ABB RobotStudio station: Session4.rspag

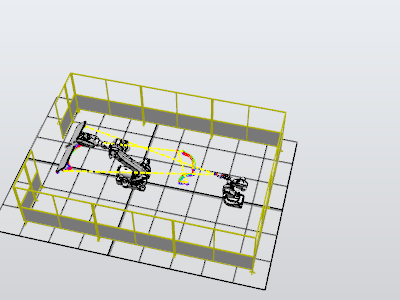
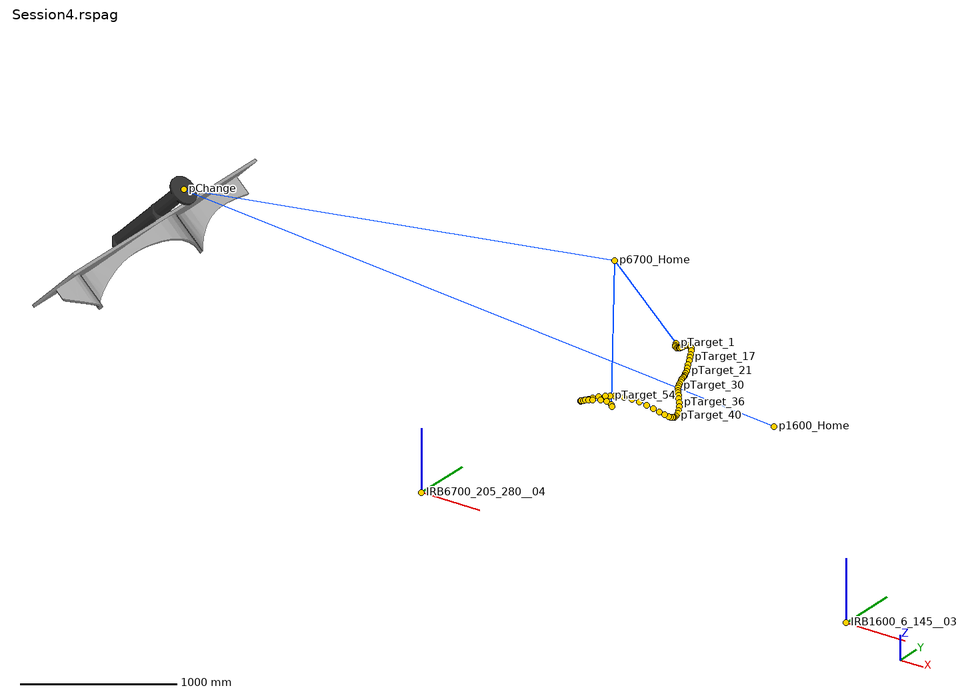
[picture v1: parts stored in the station drawn from their meshes, with robot base, taught points and paths (robot models come from the ABB library and are not in the file)]
--- station ---
Station Session4i (saved by RobotStudio 24.2.10821.1)
Controller Controller5, task T_ROB2: task frame (RAPID world) sits at (3300, 0, 0) mm, rotated rx 0 ry 0 rz 180 deg in the station
Controller Controller5, task T_ROB1: task frame (RAPID world) sits at (3300, 0, 0) mm, rotated rx 0 ry 0 rz 180 deg in the station
Controller Controller5
  mechanical unit ROB_1: IRB6700_205_280__04, 6 joints, base frame (3300, 0, 0) mm, rotated rx 0 ry 0 rz 180 deg
  mechanical unit ROB_2: IRB1600_6_145__03, 6 joints, base frame (0, 0, 0) mm
Layout (positions relative to the parent item):
  - IRB1600_6_145__03 [mechanism, from %ABB.RobotStudio.Models.IRB1600%\IRB1600_6_145_G_03.rslib] at (3300, 0, 0) mm, rotated rx 0 ry 0 rz 180 deg; joint values [0, -0.6981, 0.3491, 0, 0.4363, 3.1416] (rad or m)
  - IRB6700_205_280__04 [mechanism, from %ABB.RobotStudio.Models.IRB6700%\IRB6700_205_280__04.rslib] at (0, 0, 0) mm; joint values [0, -0.6981, -2.2689, 0, -0.9599, 0] (rad or m)
  - fence [graphiccomponentgroup, from Library\fence.rslib] at (-1500, 0, 0) mm
    - Fence_2500_1 [graphiccomponentgroup, from Equipment\Fence_2500.rslib] at (6000, 0, 0) mm
      - Body 1 [part, from Equipment\Fence_2500.rslib]
      - Body 2 [part, from Equipment\Fence_2500.rslib]
    - Fence_2500_2 [graphiccomponentgroup, from Equipment\Fence_2500.rslib] at (6000, -2500, 0) mm
      - Body 1 [part, from Equipment\Fence_2500.rslib]
      - Body 2 [part, from Equipment\Fence_2500.rslib]
    - Fence_2500_3 [graphiccomponentgroup, from Equipment\Fence_2500.rslib] at (6000, 2500, 0) mm, rotated rx 0 ry 0 rz 90 deg
      - Body 1 [part, from Equipment\Fence_2500.rslib]
      - Body 2 [part, from Equipment\Fence_2500.rslib]
    - Fence_2500_4 [graphiccomponentgroup, from Equipment\Fence_2500.rslib] at (6000, -2500, 0) mm, rotated rx 0 ry 0 rz 90 deg
      - Body 1 [part, from Equipment\Fence_2500.rslib]
      - Body 2 [part, from Equipment\Fence_2500.rslib]
    - Fence_2500_5 [graphiccomponentgroup, from Equipment\Fence_2500.rslib] at (3500, 2500, 0) mm, rotated rx 0 ry 0 rz 90 deg
      - Body 1 [part, from Equipment\Fence_2500.rslib]
      - Body 2 [part, from Equipment\Fence_2500.rslib]
    - Fence_2500_6 [graphiccomponentgroup, from Equipment\Fence_2500.rslib] at (3500, -2500, 0) mm, rotated rx 0 ry 0 rz 90 deg
      - Body 1 [part, from Equipment\Fence_2500.rslib]
      - Body 2 [part, from Equipment\Fence_2500.rslib]
    - Fence_2500_7 [graphiccomponentgroup, from Equipment\Fence_2500.rslib] at (1000, -2500, 0) mm, rotated rx 0 ry 0 rz 90 deg
      - Body 1 [part, from Equipment\Fence_2500.rslib]
      - Body 2 [part, from Equipment\Fence_2500.rslib]
    - Fence_2500_8 [graphiccomponentgroup, from Equipment\Fence_2500.rslib] at (1000, 2500, 0) mm, rotated rx 0 ry 0 rz 90 deg
      - Body 1 [part, from Equipment\Fence_2500.rslib]
      - Body 2 [part, from Equipment\Fence_2500.rslib]
    - Fence_Gate [graphiccomponentgroup, from Equipment\Fence_Gate.rslib] at (-1500, 2500, 0) mm, rotated rx 0 ry 0 rz 180 deg
      - Body 1 [part, from Equipment\Fence_Gate.rslib]
      - Body 2 [part, from Equipment\Fence_Gate.rslib]
      - Body 3 [part, from Equipment\Fence_Gate.rslib]
    - Fence_Gate_1 [graphiccomponentgroup, from Equipment\Fence_Gate.rslib] at (-1500, -1040, 0) mm, rotated rx 0 ry 0 rz 180 deg
      - Body 1 [part, from Equipment\Fence_Gate.rslib]
      - Body 2 [part, from Equipment\Fence_Gate.rslib]
      - Body 3 [part, from Equipment\Fence_Gate.rslib]
  - mySpintecTool [mechanism, from Library\mySpintecTool.rslib] at (2971.38, 0, 1222.28) mm, rotated rx -180 ry -85 rz 180 deg
  - training_part1 [part] at (-1843.45, 0, 1627.49) mm, rotated rx 180 ry -45 rz 180 deg, size 449.3 x 2022.8 x 720 mm
Attachment: mySpintecTool is attached to IRB1600_6_145__03 / Link6
Attachment: training_part1 is attached to IRB6700_205_280__04 / Link6
Targets, tools, work objects and paths stored in the station and not in the controller backup, written as RAPID:
! task T_ROB1
MODULE Module1
  VAR SyncIdent Ident_1;
  VAR SyncIdent Ident_2;
ENDMODULE

! task T_ROB2
MODULE Module1
  CONST robtarget Target_10:=[[-249.999367219,-2.759503933,70.911791319],[0.082627052,-0.189001665,0.896559115,0.391960322],[0,0,0,0],[9E+09,9E+09,9E+09,9E+09,9E+09,9E+09]];
  CONST robtarget Target_20:=[[-272.860994804,33.003713337,109.273686321],[0.078888886,-0.183345526,0.900091869,0.387292639],[0,0,0,0],[9E+09,9E+09,9E+09,9E+09,9E+09,9E+09]];
  CONST robtarget Target_30:=[[-293.909747151,69.703915361,146.790608764],[0.066447689,-0.162722707,0.911372094,0.372165194],[0,0,0,0],[9E+09,9E+09,9E+09,9E+09,9E+09,9E+09]];
  CONST robtarget Target_40:=[[-309.049057288,104.287364252,178.817535141],[0.044488261,-0.119397612,0.929423604,0.346318884],[0,0,0,0],[9E+09,9E+09,9E+09,9E+09,9E+09,9E+09]];
  CONST robtarget Target_50:=[[-315.82436696,131.079185384,200.514549492],[0.018847209,-0.056496391,0.946916759,0.315913899],[0,0,0,0],[9E+09,9E+09,9E+09,9E+09,9E+09,9E+09]];
  CONST robtarget Target_60:=[[-316.949093873,142.442010103,208.738875508],[0.005635439,-0.017961808,0.953951582,0.299369328],[0,0,0,0],[9E+09,9E+09,9E+09,9E+09,9E+09,9E+09]];
  CONST robtarget Target_70:=[[-316.981336532,150.771457316,214.363656376],[0.00472652,-0.015856219,-0.958220782,-0.285550649],[0,0,0,0],[9E+09,9E+09,9E+09,9E+09,9E+09,9E+09]];
  CONST robtarget Target_80:=[[-316.204048535,159.553535577,219.906336386],[0.015917508,-0.05682374,-0.961261763,-0.269246205],[0,0,0,0],[9E+09,9E+09,9E+09,9E+09,9E+09,9E+09]];
  CONST robtarget Target_90:=[[-312.751266422,174.803616127,228.540118146],[0.032209123,-0.130949879,-0.962189752,-0.236654987],[0,0,0,0],[9E+09,9E+09,9E+09,9E+09,9E+09,9E+09]];
  CONST robtarget Target_100:=[[-304.928487553,193.590972725,237.35167523],[0.043068547,-0.216929266,-0.956567695,-0.189907974],[0,0,0,0],[9E+09,9E+09,9E+09,9E+09,9E+09,9E+09]];
  CONST robtarget Target_110:=[[-295.35254505,209.582414865,243.17789314],[0.042988124,-0.279779228,-0.947977395,-0.145651859],[0,0,0,0],[9E+09,9E+09,9E+09,9E+09,9E+09,9E+09]];
  CONST robtarget Target_120:=[[-283.89767317,224.89172178,247.2508217],[0.035173025,-0.328290116,-0.938550871,-0.100552084],[0,0,0,0],[9E+09,9E+09,9E+09,9E+09,9E+09,9E+09]];
  CONST robtarget Target_130:=[[-263.239275575,247.748070357,250.552666299],[0.014250971,-0.37796017,-0.925055022,-0.034874436],[0,0,0,0],[9E+09,9E+09,9E+09,9E+09,9E+09,9E+09]];
  CONST robtarget Target_140:=[[-240.980203403,269.118585414,250.90982541],[0.007976683,0.402341156,0.915275131,-0.018149404],[0,0,0,0],[9E+09,9E+09,9E+09,9E+09,9E+09,9E+09]];
  CONST robtarget Target_150:=[[-208.411538431,298.031041245,247.790506063],[0.034910793,0.408676536,0.908701592,-0.077628235],[0,0,0,0],[9E+09,9E+09,9E+09,9E+09,9E+09,9E+09]];
  CONST robtarget Target_160:=[[-176.050652943,326.808930331,241.226021251],[0.053503703,0.389404955,0.910952455,-0.125166922],[0,0,0,0],[9E+09,9E+09,9E+09,9E+09,9E+09,9E+09]];
  CONST robtarget Target_170:=[[-156.251547721,345.811133404,235.321691527],[0.059919365,0.36278175,0.917514208,-0.151547844],[0,0,0,0],[9E+09,9E+09,9E+09,9E+09,9E+09,9E+09]];
  CONST robtarget Target_180:=[[-137.911367006,365.728959049,228.015632898],[0.060848306,0.321409713,0.928490022,-0.175782705],[0,0,0,0],[9E+09,9E+09,9E+09,9E+09,9E+09,9E+09]];
  CONST robtarget Target_190:=[[-123.074825841,385.296017373,219.901370788],[0.055303407,0.265093219,0.942346679,-0.196595667],[0,0,0,0],[9E+09,9E+09,9E+09,9E+09,9E+09,9E+09]];
  CONST robtarget Target_200:=[[-112.483952008,403.752551203,211.51909834],[0.044543145,0.199537763,0.95536135,-0.213272783],[0,0,0,0],[9E+09,9E+09,9E+09,9E+09,9E+09,9E+09]];
  CONST robtarget Target_210:=[[-105.66911776,420.539983076,203.415477486],[0.032817077,0.140384123,0.963573356,-0.225259238],[0,0,0,0],[9E+09,9E+09,9E+09,9E+09,9E+09,9E+09]];
  CONST robtarget Target_220:=[[-101.152730173,437.795026941,194.70341226],[0.02007137,0.08291124,0.968380047,-0.234441785],[0,0,0,0],[9E+09,9E+09,9E+09,9E+09,9E+09,9E+09]];
  CONST robtarget Target_230:=[[-99.0040493,453.549567144,186.489814416],[0.008561695,0.034579383,0.970065446,-0.240216557],[0,0,0,0],[9E+09,9E+09,9E+09,9E+09,9E+09,9E+09]];
  CONST robtarget Target_240:=[[-98.516394989,465.109909633,180.348088014],[0.000491395,0.001966291,0.970025575,-0.242994396],[0,0,0,0],[9E+09,9E+09,9E+09,9E+09,9E+09,9E+09]];
  CONST robtarget Target_250:=[[-98.913820285,477.215623072,173.84543664],[0.007456826,0.029529533,-0.969123936,0.244685919],[0,0,0,0],[9E+09,9E+09,9E+09,9E+09,9E+09,9E+09]];
  CONST robtarget Target_260:=[[-101.158760793,495.694459859,163.84647429],[0.018390599,0.072530228,-0.966611976,0.245076395],[0,0,0,0],[9E+09,9E+09,9E+09,9E+09,9E+09,9E+09]];
  CONST robtarget Target_270:=[[-106.104979829,517.566463562,152.024862353],[0.029263347,0.116194115,-0.962734999,0.242453924],[0,0,0,0],[9E+09,9E+09,9E+09,9E+09,9E+09,9E+09]];
  CONST robtarget Target_280:=[[-113.660346961,540.614341097,139.758405519],[0.038221783,0.154953239,-0.958456095,0.236411725],[0,0,0,0],[9E+09,9E+09,9E+09,9E+09,9E+09,9E+09]];
  CONST robtarget Target_290:=[[-130.507549693,578.661351825,120.440667817],[0.047524101,0.206136989,-0.952386495,0.2195654],[0,0,0,0],[9E+09,9E+09,9E+09,9E+09,9E+09,9E+09]];
  CONST robtarget Target_300:=[[-151.266393323,615.999238015,103.277260281],[0.050249688,0.24477104,-0.948497911,0.194714713],[0,0,0,0],[9E+09,9E+09,9E+09,9E+09,9E+09,9E+09]];
  CONST robtarget Target_310:=[[-176.02610459,654.710741932,88.198539481],[0.046456986,0.275583142,-0.946795556,0.159605309],[0,0,0,0],[9E+09,9E+09,9E+09,9E+09,9E+09,9E+09]];
  CONST robtarget Target_320:=[[-202.970542535,693.300547015,76.716257128],[0.035884116,0.297986116,-0.947053887,0.114041831],[0,0,0,0],[9E+09,9E+09,9E+09,9E+09,9E+09,9E+09]];
  CONST robtarget Target_330:=[[-231.602130589,732.417304287,69.542021834],[0.018589095,0.31143545,-0.948397291,0.056612584],[0,0,0,0],[9E+09,9E+09,9E+09,9E+09,9E+09,9E+09]];
  CONST robtarget Target_340:=[[-260.470210824,771.255251336,67.256102726],[0.000027118,0.313521967,-0.949580944,0.000077659],[0,0,0,0],[9E+09,9E+09,9E+09,9E+09,9E+09,9E+09]];
  CONST robtarget Target_350:=[[-291.671653455,813.968299538,69.78080258],[0.017514958,-0.303598774,0.9510575,0.054869325],[0,0,0,0],[9E+09,9E+09,9E+09,9E+09,9E+09,9E+09]];
  CONST robtarget Target_360:=[[-321.100482584,856.495332628,76.875137674],[0.030055142,-0.282317538,0.953462043,0.101506791],[0,0,0,0],[9E+09,9E+09,9E+09,9E+09,9E+09,9E+09]];
  CONST robtarget Target_370:=[[-347.608236851,898.755866406,87.798617829],[0.03661292,-0.250273308,0.957292518,0.140049279],[0,0,0,0],[9E+09,9E+09,9E+09,9E+09,9E+09,9E+09]];
  CONST robtarget Target_380:=[[-370.0464549,940.669416672,101.810752862],[0.036758138,-0.206846372,0.962600213,0.171067961],[0,0,0,0],[9E+09,9E+09,9E+09,9E+09,9E+09,9E+09]];
  CONST robtarget Target_390:=[[-386.422870207,979.737745125,117.176024402],[0.030820624,-0.15395644,0.968381142,0.193869719],[0,0,0,0],[9E+09,9E+09,9E+09,9E+09,9E+09,9E+09]];
  CONST robtarget Target_400:=[[-397.441727713,1019.682361901,134.633461354],[0.01837918,-0.084776151,0.973609592,0.211091382],[0,0,0,0],[9E+09,9E+09,9E+09,9E+09,9E+09,9E+09]];
  CONST robtarget Target_410:=[[-400.68526788,1043.112626972,145.490242444],[0.008067365,-0.036072035,0.975216982,0.218141154],[0,0,0,0],[9E+09,9E+09,9E+09,9E+09,9E+09,9E+09]];
  CONST robtarget Target_420:=[[-401.329476368,1057.285914809,152.218968855],[0.000811987,-0.00358584,0.975219049,0.221210962],[0,0,0,0],[9E+09,9E+09,9E+09,9E+09,9E+09,9E+09]];
  CONST robtarget Target_430:=[[-400.962720054,1070.625724022,158.636236091],[0.006312666,-0.02754754,-0.974356125,-0.223229532],[0,0,0,0],[9E+09,9E+09,9E+09,9E+09,9E+09,9E+09]];
  CONST robtarget Target_440:=[[-398.849530954,1089.506582954,167.817808857],[0.016104926,-0.069657841,-0.97181004,-0.224663442],[0,0,0,0],[9E+09,9E+09,9E+09,9E+09,9E+09,9E+09]];
  CONST robtarget Target_450:=[[-394.29581823,1110.83283784,178.260483341],[0.026405516,-0.113854454,-0.967470561,-0.224367166],[0,0,0,0],[9E+09,9E+09,9E+09,9E+09,9E+09,9E+09]];
  CONST robtarget Target_460:=[[-380.757667282,1149.008190868,196.879200033],[0.041846543,-0.182836175,-0.957495657,-0.219138923],[0,0,0,0],[9E+09,9E+09,9E+09,9E+09,9E+09,9E+09]];
  CONST robtarget Target_470:=[[-357.502548238,1192.923255868,217.60212677],[0.053666998,-0.246019085,-0.94554354,-0.206256825],[0,0,0,0],[9E+09,9E+09,9E+09,9E+09,9E+09,9E+09]];
  CONST robtarget Target_480:=[[-328.871131584,1234.786110626,235.983778233],[0.058387182,-0.291828294,-0.936135211,-0.187291352],[0,0,0,0],[9E+09,9E+09,9E+09,9E+09,9E+09,9E+09]];
  CONST robtarget Target_490:=[[-297.082202513,1274.587810161,251.518415059],[0.056709338,-0.324130465,-0.930183001,-0.162736218],[0,0,0,0],[9E+09,9E+09,9E+09,9E+09,9E+09,9E+09]];
  CONST robtarget Target_500:=[[-262.487169544,1314.071354306,264.397885002],[0.048966326,-0.346373772,-0.92759546,-0.131126548],[0,0,0,0],[9E+09,9E+09,9E+09,9E+09,9E+09,9E+09]];
  CONST robtarget Target_510:=[[-226.575198444,1353.203760165,273.991191603],[0.03530716,-0.35871904,-0.92829236,-0.091363833],[0,0,0,0],[9E+09,9E+09,9E+09,9E+09,9E+09,9E+09]];
  CONST robtarget Target_520:=[[-190.835454984,1391.952044842,279.667338403],[0.016347916,-0.360036739,-0.931834961,-0.042307189],[0,0,0,0],[9E+09,9E+09,9E+09,9E+09,9E+09,9E+09]];
  CONST robtarget Target_530:=[[-154.17832425,1433.250752389,280.669165784],[0.008033429,0.346250872,0.937854953,-0.021768907],[0,0,0,0],[9E+09,9E+09,9E+09,9E+09,9E+09,9E+09]];
  CONST robtarget Target_540:=[[-136.486757318,1454.463382029,278.844216812],[0.02093735,0.331543339,0.941332059,-0.059452467],[0,0,0,0],[9E+09,9E+09,9E+09,9E+09,9E+09,9E+09]];
  CONST robtarget Target_550:=[[-119.667994947,1475.942313909,275.183061704],[0.033064953,0.31046011,0.944668189,-0.100614324],[0,0,0,0],[9E+09,9E+09,9E+09,9E+09,9E+09,9E+09]];
  CONST robtarget Target_560:=[[-95.23421766,1510.929497189,264.90036064],[0.047328965,0.26196812,0.948558033,-0.171377746],[0,0,0,0],[9E+09,9E+09,9E+09,9E+09,9E+09,9E+09]];
  CONST robtarget Target_570:=[[-75.879163631,1544.775316833,249.92732557],[0.048387235,0.203046981,0.951330794,-0.226716385],[0,0,0,0],[9E+09,9E+09,9E+09,9E+09,9E+09,9E+09]];
  CONST robtarget Target_580:=[[-61.453751357,1578.969573233,230.891791828],[0.037712511,0.135799258,0.953915563,-0.264917773],[0,0,0,0],[9E+09,9E+09,9E+09,9E+09,9E+09,9E+09]];
  CONST robtarget Target_590:=[[-52.709355316,1614.593121608,208.283153837],[0.017684195,0.058897435,0.955941718,-0.287043189],[0,0,0,0],[9E+09,9E+09,9E+09,9E+09,9E+09,9E+09]];
  CONST robtarget Target_600:=[[-50.934699689,1632.587258186,196.277463107],[0.006063338,0.019886972,0.956307978,-0.291620979],[0,0,0,0],[9E+09,9E+09,9E+09,9E+09,9E+09,9E+09]];
  CONST robtarget Target_610:=[[-50.774421373,1647.958649082,185.919783485],[0.003455043,0.011306726,-0.956305426,0.292130371],[0,0,0,0],[9E+09,9E+09,9E+09,9E+09,9E+09,9E+09]];
  CONST robtarget Target_620:=[[-52.135096903,1666.482081789,173.506543624],[0.014073891,0.04660989,-0.956181617,0.28869735],[0,0,0,0],[9E+09,9E+09,9E+09,9E+09,9E+09,9E+09]];
  CONST robtarget Target_630:=[[-58.784165359,1700.876830889,151.380550889],[0.030261256,0.106897681,-0.956235195,0.270686891],[0,0,0,0],[9E+09,9E+09,9E+09,9E+09,9E+09,9E+09]];
  CONST robtarget Target_640:=[[-65.575026565,1722.872557128,138.384921656],[0.037454996,0.142723783,-0.956661626,0.251048954],[0,0,0,0],[9E+09,9E+09,9E+09,9E+09,9E+09,9E+09]];
  CONST robtarget Target_650:=[[-74.174240255,1744.953068342,126.651812084],[0.041515823,0.176927532,-0.957346748,0.224633675],[0,0,0,0],[9E+09,9E+09,9E+09,9E+09,9E+09,9E+09]];
  CONST robtarget Target_660:=[[-84.218309667,1766.689454041,116.699308849],[0.041788008,0.208774714,-0.958068354,0.191760032],[0,0,0,0],[9E+09,9E+09,9E+09,9E+09,9E+09,9E+09]];
  CONST robtarget Target_670:=[[-95.705744302,1788.48102753,108.594683736],[0.037739774,0.238344582,-0.958506502,0.151765791],[0,0,0,0],[9E+09,9E+09,9E+09,9E+09,9E+09,9E+09]];
  CONST robtarget Target_680:=[[-107.613651561,1808.886394545,102.938341083],[0.029652784,0.263007018,-0.958267247,0.108036583],[0,0,0,0],[9E+09,9E+09,9E+09,9E+09,9E+09,9E+09]];
  CONST robtarget Target_690:=[[-120.621960396,1829.451402306,99.309687547],[0.017514553,0.28370735,-0.956929474,0.059070827],[0,0,0,0],[9E+09,9E+09,9E+09,9E+09,9E+09,9E+09]];
  CONST robtarget Target_700:=[[-148.700181706,1869.906708876,98.057386407],[0.008453075,-0.309439943,0.950526698,0.025970423],[0,0,0,0],[9E+09,9E+09,9E+09,9E+09,9E+09,9E+09]];
  CONST robtarget Target_710:=[[-178.288124099,1909.002656836,102.934665136],[0.030003932,-0.320093123,0.942777752,0.088375719],[0,0,0,0],[9E+09,9E+09,9E+09,9E+09,9E+09,9E+09]];
  CONST robtarget Target_720:=[[-222.707062289,1964.208367066,117.387196058],[0.050888963,-0.321696598,0.933861387,0.147731248],[0,0,0,0],[9E+09,9E+09,9E+09,9E+09,9E+09,9E+09]];
  CONST robtarget Target_730:=[[-250.000100712,1997.24045093,129.048804233],[0.058217616,-0.318394383,0.930737336,0.17018736],[0,0,0,0],[9E+09,9E+09,9E+09,9E+09,9E+09,9E+09]];
  VAR SyncIdent Ident_1;
  VAR SyncIdent Ident_2;
  PROC Path_Process()
    MoveL Target_10,v200,z1,tSpintec\WObj:=obWorkpiece;
    MoveL Target_20,v200,z1,tSpintec\WObj:=obWorkpiece;
    MoveL Target_30,v200,z1,tSpintec\WObj:=obWorkpiece;
    MoveL Target_40,v200,z1,tSpintec\WObj:=obWorkpiece;
    MoveL Target_50,v200,z1,tSpintec\WObj:=obWorkpiece;
    MoveL Target_60,v200,z1,tSpintec\WObj:=obWorkpiece;
    MoveL Target_70,v200,z1,tSpintec\WObj:=obWorkpiece;
    MoveL Target_80,v200,z1,tSpintec\WObj:=obWorkpiece;
    MoveL Target_90,v200,z1,tSpintec\WObj:=obWorkpiece;
    MoveL Target_100,v200,z1,tSpintec\WObj:=obWorkpiece;
    MoveL Target_110,v200,z1,tSpintec\WObj:=obWorkpiece;
    MoveL Target_120,v200,z1,tSpintec\WObj:=obWorkpiece;
    MoveL Target_130,v200,z1,tSpintec\WObj:=obWorkpiece;
    MoveL Target_140,v200,z1,tSpintec\WObj:=obWorkpiece;
    MoveL Target_150,v200,z1,tSpintec\WObj:=obWorkpiece;
    MoveL Target_160,v200,z1,tSpintec\WObj:=obWorkpiece;
    MoveL Target_170,v200,z1,tSpintec\WObj:=obWorkpiece;
    MoveL Target_180,v200,z1,tSpintec\WObj:=obWorkpiece;
    MoveL Target_190,v200,z1,tSpintec\WObj:=obWorkpiece;
    MoveL Target_200,v200,z1,tSpintec\WObj:=obWorkpiece;
    MoveL Target_210,v200,z1,tSpintec\WObj:=obWorkpiece;
    MoveL Target_220,v200,z1,tSpintec\WObj:=obWorkpiece;
    MoveL Target_230,v200,z1,tSpintec\WObj:=obWorkpiece;
    MoveL Target_240,v200,z1,tSpintec\WObj:=obWorkpiece;
    MoveL Target_250,v200,z1,tSpintec\WObj:=obWorkpiece;
    MoveL Target_260,v200,z1,tSpintec\WObj:=obWorkpiece;
    MoveL Target_270,v200,z1,tSpintec\WObj:=obWorkpiece;
    MoveL Target_280,v200,z1,tSpintec\WObj:=obWorkpiece;
    MoveL Target_290,v200,z1,tSpintec\WObj:=obWorkpiece;
    MoveL Target_300,v200,z1,tSpintec\WObj:=obWorkpiece;
    MoveL Target_310,v200,z1,tSpintec\WObj:=obWorkpiece;
    MoveL Target_320,v200,z1,tSpintec\WObj:=obWorkpiece;
    MoveL Target_330,v200,z1,tSpintec\WObj:=obWorkpiece;
    MoveL Target_340,v200,z1,tSpintec\WObj:=obWorkpiece;
    MoveL Target_350,v200,z1,tSpintec\WObj:=obWorkpiece;
    MoveL Target_360,v200,z1,tSpintec\WObj:=obWorkpiece;
    MoveL Target_370,v200,z1,tSpintec\WObj:=obWorkpiece;
    MoveL Target_380,v200,z1,tSpintec\WObj:=obWorkpiece;
    MoveL Target_390,v200,z1,tSpintec\WObj:=obWorkpiece;
    MoveL Target_400,v200,z1,tSpintec\WObj:=obWorkpiece;
    MoveL Target_410,v200,z1,tSpintec\WObj:=obWorkpiece;
    MoveL Target_420,v200,z1,tSpintec\WObj:=obWorkpiece;
    MoveL Target_430,v200,z1,tSpintec\WObj:=obWorkpiece;
    MoveL Target_440,v200,z1,tSpintec\WObj:=obWorkpiece;
    MoveL Target_450,v200,z1,tSpintec\WObj:=obWorkpiece;
    MoveL Target_460,v200,z1,tSpintec\WObj:=obWorkpiece;
    MoveL Target_470,v200,z1,tSpintec\WObj:=obWorkpiece;
    MoveL Target_480,v200,z1,tSpintec\WObj:=obWorkpiece;
    MoveL Target_490,v200,z1,tSpintec\WObj:=obWorkpiece;
    MoveL Target_500,v200,z1,tSpintec\WObj:=obWorkpiece;
    MoveL Target_510,v200,z1,tSpintec\WObj:=obWorkpiece;
    MoveL Target_520,v200,z1,tSpintec\WObj:=obWorkpiece;
    MoveL Target_530,v200,z1,tSpintec\WObj:=obWorkpiece;
    MoveL Target_540,v200,z1,tSpintec\WObj:=obWorkpiece;
    MoveL Target_550,v200,z1,tSpintec\WObj:=obWorkpiece;
    MoveL Target_560,v200,z1,tSpintec\WObj:=obWorkpiece;
    MoveL Target_570,v200,z1,tSpintec\WObj:=obWorkpiece;
    MoveL Target_580,v200,z1,tSpintec\WObj:=obWorkpiece;
    MoveL Target_590,v200,z1,tSpintec\WObj:=obWorkpiece;
    MoveL Target_600,v200,z1,tSpintec\WObj:=obWorkpiece;
    MoveL Target_610,v200,z1,tSpintec\WObj:=obWorkpiece;
    MoveL Target_620,v200,z1,tSpintec\WObj:=obWorkpiece;
    MoveL Target_630,v200,z1,tSpintec\WObj:=obWorkpiece;
    MoveL Target_640,v200,z1,tSpintec\WObj:=obWorkpiece;
    MoveL Target_650,v200,z1,tSpintec\WObj:=obWorkpiece;
    MoveL Target_660,v200,z1,tSpintec\WObj:=obWorkpiece;
    MoveL Target_670,v200,z1,tSpintec\WObj:=obWorkpiece;
    MoveL Target_680,v200,z1,tSpintec\WObj:=obWorkpiece;
    MoveL Target_690,v200,z1,tSpintec\WObj:=obWorkpiece;
    MoveL Target_700,v200,z1,tSpintec\WObj:=obWorkpiece;
    MoveL Target_710,v200,z1,tSpintec\WObj:=obWorkpiece;
    MoveL Target_720,v200,z1,tSpintec\WObj:=obWorkpiece;
    MoveL Target_730,v200,z1,tSpintec\WObj:=obWorkpiece;
  ENDPROC
ENDMODULE


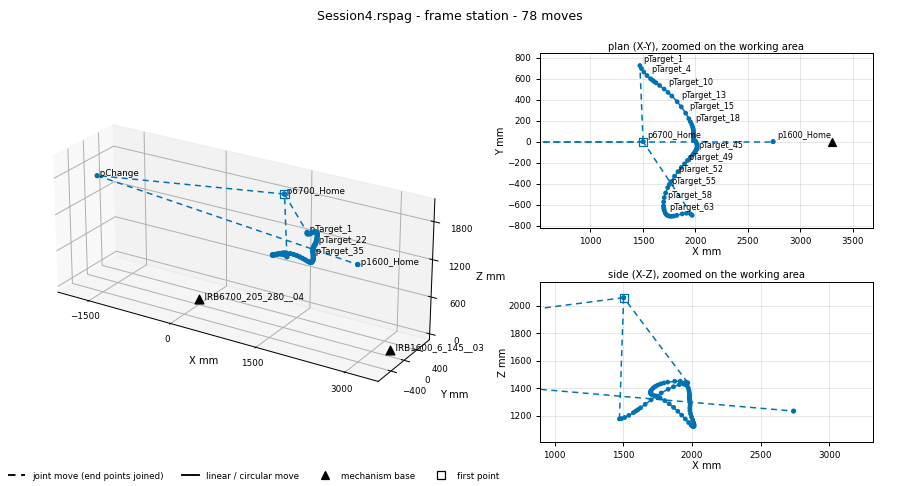
[picture p0: tool path of Session4.rspag in frame station, 78 of 151 moves have a stored position in this frame; points joined in program order, loops and branches not executed]
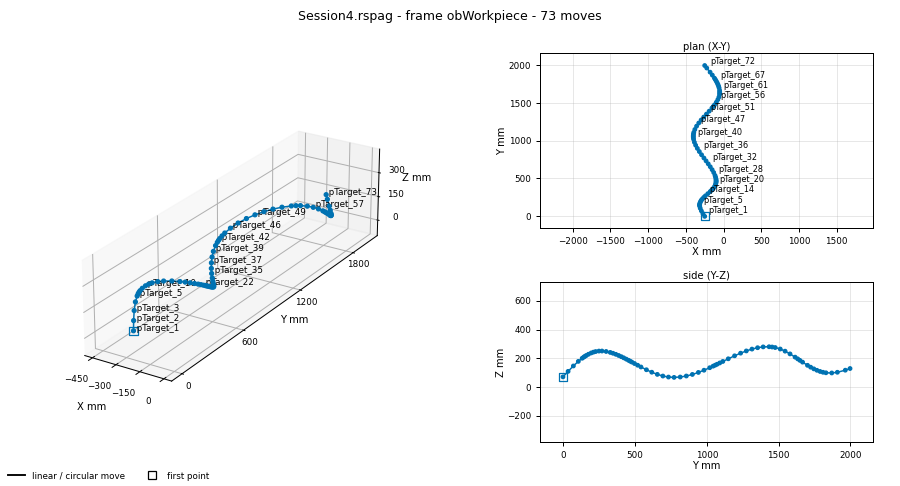
[picture p1: tool path of Session4.rspag in frame obWorkpiece, 73 of 151 moves have a stored position in this frame; points joined in program order, loops and branches not executed]
--- Backups/Controller5/RAPID/TASK1/PROGMOD/Module1.mod ---
MODULE Module1
        CONST robtarget p6700_Home:=[[1797.5,0,2060],[0,1,0,0],[0,0,0,0],[9E+09,9E+09,9E+09,9E+09,9E+09,9E+09]];
    VAR syncident Ident_1;
    PERS tasks Task_1{2}:=[["T_ROB1"],["T_ROB2"]];
    CONST robtarget pTarget_1:=[[1828.284203915,-724.31168321,1177.13895727],[0.178676959,-0.894088998,-0.396772871,-0.106069301],[0,-1,-1,0],[9E+09,9E+09,9E+09,9E+09,9E+09,9E+09]];
    CONST robtarget pTarget_2:=[[1813.352283995,-695.466433506,1178.773420247],[0.17610781,-0.899414857,-0.385704383,-0.106165355],[0,-1,-1,0],[9E+09,9E+09,9E+09,9E+09,9E+09,9E+09]];
    CONST robtarget pTarget_3:=[[1790.906859407,-662.976610401,1186.91351966],[0.166255441,-0.909877659,-0.366663235,-0.100199034],[0,-1,-1,0],[9E+09,9E+09,9E+09,9E+09,9E+09,9E+09]];
    CONST robtarget pTarget_4:=[[1760.343096017,-628.860180936,1202.462053021],[0.146821719,-0.925365456,-0.33859941,-0.086559777],[0,-1,-1,0],[9E+09,9E+09,9E+09,9E+09,9E+09,9E+09]];
    CONST robtarget pTarget_5:=[[1726.254200272,-598.401420489,1222.697580978],[0.120661974,-0.941940185,-0.305967435,-0.067626216],[0,-1,-1,0],[9E+09,9E+09,9E+09,9E+09,9E+09,9E+09]];
    CONST robtarget pTarget_6:=[[1707.760831936,-583.808712968,1234.618090687],[0.105401093,-0.950166225,-0.287900298,-0.0564639],[0,-1,-1,0],[9E+09,9E+09,9E+09,9E+09,9E+09,9E+09]];
    CONST robtarget pTarget_7:=[[1692.345626917,-572.272275695,1245.084662397],[0.092337209,-0.956523353,-0.272660527,-0.046831106],[0,-1,-1,0],[9E+09,9E+09,9E+09,9E+09,9E+09,9E+09]];
    CONST robtarget pTarget_8:=[[1674.311096497,-559.259450538,1258.017005989],[0.076818082,-0.963341264,-0.254613251,-0.035280078],[0,-1,-1,0],[9E+09,9E+09,9E+09,9E+09,9E+09,9E+09]];
    CONST robtarget pTarget_9:=[[1640.749420506,-534.675686209,1283.12739558],[0.0488623,-0.974033719,-0.220623448,-0.014002965],[0,-1,-1,0],[9E+09,9E+09,9E+09,9E+09,9E+09,9E+09]];
    CONST robtarget pTarget_10:=[[1597.548085701,-500.707722699,1315.809510935],[0.015723588,-0.984093125,-0.176553972,0.011924134],[0,-1,-1,0],[9E+09,9E+09,9E+09,9E+09,9E+09,9E+09]];
    CONST robtarget pTarget_11:=[[1560.122160725,-468.232280243,1342.630652695],[0.009960351,0.989770979,0.138573814,-0.032426835],[0,0,-1,0],[9E+09,9E+09,9E+09,9E+09,9E+09,9E+09]];
    CONST robtarget pTarget_12:=[[1524.075108455,-433.938166023,1365.597259362],[0.031800185,0.99294942,0.102617389,-0.050098597],[0,0,-1,0],[9E+09,9E+09,9E+09,9E+09,9E+09,9E+09]];
    CONST robtarget pTarget_13:=[[1473.522255972,-380.040760556,1393.007827396],[0.058309144,0.994274382,0.053111798,-0.072094615],[0,0,0,0],[9E+09,9E+09,9E+09,9E+09,9E+09,9E+09]];
    CONST robtarget pTarget_14:=[[1434.168369928,-331.47546633,1411.352090434],[0.07596009,0.993123055,0.014704628,-0.087866016],[0,0,0,0],[9E+09,9E+09,9E+09,9E+09,9E+09,9E+09]];
    CONST robtarget pTarget_15:=[[1392.526878043,-271.019237865,1426.398673898],[0.090329873,0.990180936,-0.025534371,-0.10358679],[0,0,0,0],[9E+09,9E+09,9E+09,9E+09,9E+09,9E+09]];
    CONST robtarget pTarget_16:=[[1362.239039529,-218.541069015,1430.539167166],[0.094666583,0.987515076,-0.052742603,-0.114325982],[0,0,0,0],[9E+09,9E+09,9E+09,9E+09,9E+09,9E+09]];
    CONST robtarget pTarget_17:=[[1347.116933407,-188.685960016,1426.792004509],[0.092012599,0.986546292,-0.063605198,-0.11922447],[0,0,0,0],[9E+09,9E+09,9E+09,9E+09,9E+09,9E+09]];
    CONST robtarget pTarget_18:=[[1334.819790939,-161.863170399,1416.798445755],[0.084118359,0.986498153,-0.068454591,-0.122717013],[0,0,0,0],[9E+09,9E+09,9E+09,9E+09,9E+09,9E+09]];
    CONST robtarget pTarget_19:=[[1326.354610986,-140.212828624,1400.977626515],[0.070776066,0.987462113,-0.065959344,-0.124734471],[0,0,0,0],[9E+09,9E+09,9E+09,9E+09,9E+09,9E+09]];
    CONST robtarget pTarget_20:=[[1321.900977392,-123.747496931,1382.919237529],[0.053938466,0.988914891,-0.057413339,-0.125863771],[0,0,0,0],[9E+09,9E+09,9E+09,9E+09,9E+09,9E+09]];
    CONST robtarget pTarget_21:=[[1319.886923651,-110.789994279,1368.508392884],[0.038480736,0.990002275,-0.047766182,-0.127016222],[0,0,0,0],[9E+09,9E+09,9E+09,9E+09,9E+09,9E+09]];
    CONST robtarget pTarget_22:=[[1319.175199159,-98.828778796,1356.427746111],[0.023312333,0.990748793,-0.037113612,-0.128436536],[0,0,0,0],[9E+09,9E+09,9E+09,9E+09,9E+09,9E+09]];
    CONST robtarget pTarget_23:=[[1319.187042676,-88.760210155,1347.718921985],[0.010438451,0.991093279,-0.027321467,-0.129918003],[0,0,0,0],[9E+09,9E+09,9E+09,9E+09,9E+09,9E+09]];
    CONST robtarget pTarget_24:=[[1319.345634363,-81.767119465,1342.525728764],[0.001666911,0.991162936,-0.020300956,-0.131076801],[0,-1,0,0],[9E+09,9E+09,9E+09,9E+09,9E+09,9E+09]];
    CONST robtarget pTarget_25:=[[1319.500322179,-74.746781592,1337.952171624],[0.006900487,-0.99109643,0.013182328,0.13231204],[0,-1,0,0],[9E+09,9E+09,9E+09,9E+09,9E+09,9E+09]];
    CONST robtarget pTarget_26:=[[1319.527904378,-64.575839297,1332.207735248],[0.018834765,-0.990778505,0.002817167,0.134146447],[0,-1,0,0],[9E+09,9E+09,9E+09,9E+09,9E+09,9E+09]];
    CONST robtarget pTarget_27:=[[1319.092832552,-53.386463681,1326.571421044],[0.031412834,-0.990161471,-0.008772728,0.13607547],[0,-1,0,0],[9E+09,9E+09,9E+09,9E+09,9E+09,9E+09]];
    CONST robtarget pTarget_28:=[[1318.125198056,-42.651848538,1321.164194853],[0.043248684,-0.989324138,-0.020505123,0.137647527],[0,-1,0,0],[9E+09,9E+09,9E+09,9E+09,9E+09,9E+09]];
    CONST robtarget pTarget_29:=[[1315.949151126,-27.634884312,1311.998611575],[0.060671906,-0.987646517,-0.03989292,0.138859038],[0,-1,0,0],[9E+09,9E+09,9E+09,9E+09,9E+09,9E+09]];
    CONST robtarget pTarget_30:=[[1314.047443313,-16.722015814,1301.681897871],[0.076384349,-0.985616767,-0.060422194,0.138109298],[0,-1,0,0],[9E+09,9E+09,9E+09,9E+09,9E+09,9E+09]];
    CONST robtarget pTarget_31:=[[1313.24780987,-10.107768229,1289.112209707],[0.092144011,-0.982893956,-0.084701348,0.135109713],[0,-1,0,0],[9E+09,9E+09,9E+09,9E+09,9E+09,9E+09]];
    CONST robtarget pTarget_32:=[[1314.061557744,-8.924296392,1274.355069955],[0.107748776,-0.97918154,-0.112929836,0.129771206],[0,-1,-1,0],[9E+09,9E+09,9E+09,9E+09,9E+09,9E+09]];
    CONST robtarget pTarget_33:=[[1316.122761118,-13.272956057,1256.717019544],[0.123250709,-0.974011426,-0.145618271,0.122091458],[0,-1,-1,0],[9E+09,9E+09,9E+09,9E+09,9E+09,9E+09]];
    CONST robtarget pTarget_34:=[[1315.287165692,-16.436218207,1236.993976149],[0.135474574,-0.968600291,-0.174496533,0.114066107],[0,-1,-1,0],[9E+09,9E+09,9E+09,9E+09,9E+09,9E+09]];
    CONST robtarget pTarget_35:=[[1310.397078609,-15.0041594,1214.08369893],[0.144251948,-0.963620749,-0.19837115,0.106185285],[0,-1,-1,0],[9E+09,9E+09,9E+09,9E+09,9E+09,9E+09]];
    CONST robtarget pTarget_36:=[[1303.055638332,-8.361206787,1191.251607332],[0.148437826,-0.96032919,-0.21390481,0.099893899],[0,-1,-1,0],[9E+09,9E+09,9E+09,9E+09,9E+09,9E+09]];
    CONST robtarget pTarget_37:=[[1295.086167147,3.014803047,1169.686949622],[0.148305338,-0.959111684,-0.22131092,0.095560347],[0,-1,-1,0],[9E+09,9E+09,9E+09,9E+09,9E+09,9E+09]];
    CONST robtarget pTarget_38:=[[1288.230526453,18.305545049,1150.463747846],[0.143927978,-0.960119234,-0.2207257,0.093466356],[0,-1,-1,0],[9E+09,9E+09,9E+09,9E+09,9E+09,9E+09]];
    CONST robtarget pTarget_39:=[[1284.302335445,35.363619178,1135.570148534],[0.135802691,-0.963055702,-0.212787276,0.093823867],[0,-1,-1,0],[9E+09,9E+09,9E+09,9E+09,9E+09,9E+09]];
    CONST robtarget pTarget_40:=[[1284.354511494,54.631681113,1124.996395155],[0.123120654,-0.96783909,-0.196804372,0.096937294],[-1,-1,-1,0],[9E+09,9E+09,9E+09,9E+09,9E+09,9E+09]];
    CONST robtarget pTarget_41:=[[1287.005761171,66.320152526,1121.9879587],[0.113546866,-0.971262994,-0.183574805,0.100277598],[-1,-1,-1,0],[9E+09,9E+09,9E+09,9E+09,9E+09,9E+09]];
    CONST robtarget pTarget_42:=[[1289.739794546,73.372765689,1121.691299889],[0.107018008,-0.973453554,-0.17420622,0.102895663],[-1,-1,-1,0],[9E+09,9E+09,9E+09,9E+09,9E+09,9E+09]];
    CONST robtarget pTarget_43:=[[1293.076244267,80.02005922,1122.681655716],[0.100743717,-0.975448097,-0.164896007,0.105645729],[-1,-1,-1,0],[9E+09,9E+09,9E+09,9E+09,9E+09,9E+09]];
    CONST robtarget pTarget_44:=[[1298.881611111,89.612751558,1126.19063305],[0.092307855,-0.977967676,-0.151728228,0.109713394],[-1,-1,-1,0],[9E+09,9E+09,9E+09,9E+09,9E+09,9E+09]];
    CONST robtarget pTarget_45:=[[1306.820556835,100.792917172,1132.790637794],[0.083497957,-0.980382795,-0.137063638,0.114416897],[-1,-1,-1,0],[9E+09,9E+09,9E+09,9E+09,9E+09,9E+09]];
    CONST robtarget pTarget_46:=[[1324.182190694,122.110889916,1150.157313827],[0.069703098,-0.98367019,-0.111696188,0.122712662],[-1,-1,-1,0],[9E+09,9E+09,9E+09,9E+09,9E+09,9E+09]];
    CONST robtarget pTarget_47:=[[1348.359608615,149.461188423,1176.202467534],[0.056598622,-0.986147273,-0.083692311,0.131551319],[-1,-1,-1,0],[9E+09,9E+09,9E+09,9E+09,9E+09,9E+09]];
    CONST robtarget pTarget_48:=[[1375.046822103,179.052522554,1204.5172307],[0.046087562,-0.987562933,-0.057187212,0.139014431],[-1,-1,-1,0],[9E+09,9E+09,9E+09,9E+09,9E+09,9E+09]];
    CONST robtarget pTarget_49:=[[1403.348248008,210.846930482,1232.803088455],[0.037155801,-0.988221872,-0.03102722,0.145169868],[-1,-1,-1,0],[9E+09,9E+09,9E+09,9E+09,9E+09,9E+09]];
    CONST robtarget pTarget_50:=[[1433.866942492,246.305159921,1260.74682538],[0.028760176,-0.988210729,-0.003129686,0.150341652],[-1,-1,-1,0],[9E+09,9E+09,9E+09,9E+09,9E+09,9E+09]];
    CONST robtarget pTarget_51:=[[1465.920152931,285.671375259,1286.965690906],[0.020560355,-0.987398943,0.027238607,0.154527203],[-1,-1,-1,0],[9E+09,9E+09,9E+09,9E+09,9E+09,9E+09]];
    CONST robtarget pTarget_52:=[[1498.449404024,329.107412865,1310.075465317],[0.012534259,-0.985546949,0.060397799,0.157772649],[-1,0,-1,0],[9E+09,9E+09,9E+09,9E+09,9E+09,9E+09]];
    CONST robtarget pTarget_53:=[[1532.214887428,380.391805224,1329.998200772],[0.004590641,-0.982072514,0.09880022,0.16047124],[-1,0,-1,0],[9E+09,9E+09,9E+09,9E+09,9E+09,9E+09]];
    CONST robtarget pTarget_54:=[[1548.365312984,408.62004815,1337.877486917],[0.001149172,-0.979592308,0.119273236,0.161776033],[-1,0,-1,0],[9E+09,9E+09,9E+09,9E+09,9E+09,9E+09]];
    CONST robtarget pTarget_55:=[[1563.343327182,438.339613113,1344.106539286],[0.001568625,0.976592662,-0.140032512,-0.163264223],[-1,0,-1,0],[9E+09,9E+09,9E+09,9E+09,9E+09,9E+09]];
    CONST robtarget pTarget_56:=[[1583.572451273,488.207987388,1350.845108015],[0.003415808,0.970879459,-0.171981466,-0.166744668],[-1,0,0,0],[9E+09,9E+09,9E+09,9E+09,9E+09,9E+09]];
    CONST robtarget pTarget_57:=[[1595.961150028,532.687698502,1356.158800395],[0.000927714,-0.966089132,0.192044342,0.172597504],[-1,0,0,0],[9E+09,9E+09,9E+09,9E+09,9E+09,9E+09]];
    CONST robtarget pTarget_58:=[[1602.127130867,573.173660699,1362.420286483],[0.011475127,-0.962754926,0.200323018,0.181223514],[-1,0,0,0],[9E+09,9E+09,9E+09,9E+09,9E+09,9E+09]];
    CONST robtarget pTarget_59:=[[1602.651896047,611.552890659,1371.059967122],[0.028132379,-0.960699101,0.197657455,0.192866112],[-1,-1,0,0],[9E+09,9E+09,9E+09,9E+09,9E+09,9E+09]];
    CONST robtarget pTarget_60:=[[1600.989132007,629.279466214,1376.344004429],[0.037922464,-0.960007936,0.192886852,0.199352233],[-1,-1,0,0],[9E+09,9E+09,9E+09,9E+09,9E+09,9E+09]];
    CONST robtarget pTarget_61:=[[1598.81256338,643.244408001,1381.175023796],[0.046401065,-0.959519146,0.18766468,0.204821674],[-1,-1,0,0],[9E+09,9E+09,9E+09,9E+09,9E+09,9E+09]];
    CONST robtarget pTarget_62:=[[1595.17441565,658.630987476,1387.299264521],[0.056819148,-0.95903726,0.179933633,0.211288915],[-1,-1,0,0],[9E+09,9E+09,9E+09,9E+09,9E+09,9E+09]];
    CONST robtarget pTarget_63:=[[1584.898557649,682.840453061,1399.377104364],[0.077051939,-0.958365217,0.161016617,0.222873864],[-1,-1,0,0],[9E+09,9E+09,9E+09,9E+09,9E+09,9E+09]];
    CONST robtarget pTarget_64:=[[1575.343369548,695.014578464,1407.468394705],[0.090823591,-0.957971138,0.145400422,0.230002374],[-1,-1,0,0],[9E+09,9E+09,9E+09,9E+09,9E+09,9E+09]];
    CONST robtarget pTarget_65:=[[1562.790581344,704.184776879,1415.785137358],[0.105437903,-0.957458593,0.126599701,0.236914347],[-1,-1,0,0],[9E+09,9E+09,9E+09,9E+09,9E+09,9E+09]];
    CONST robtarget pTarget_66:=[[1546.931319762,709.699336183,1423.998266342],[0.120623037,-0.956665453,0.104787205,0.24343569],[-1,-1,-1,0],[9E+09,9E+09,9E+09,9E+09,9E+09,9E+09]];
    CONST robtarget pTarget_67:=[[1526.911194813,711.116279427,1431.971910731],[0.136559726,-0.955362564,0.079513962,0.249622401],[-1,-1,-1,0],[9E+09,9E+09,9E+09,9E+09,9E+09,9E+09]];
    CONST robtarget pTarget_68:=[[1503.949403484,708.1842678,1438.837208394],[0.15194001,-0.95345797,0.052864779,0.255024405],[-1,-1,-1,0],[9E+09,9E+09,9E+09,9E+09,9E+09,9E+09]];
    CONST robtarget pTarget_69:=[[1476.829540839,701.058601123,1444.688802896],[0.167442415,-0.950684259,0.023883487,0.259984723],[-1,-1,-1,0],[9E+09,9E+09,9E+09,9E+09,9E+09,9E+09]];
    CONST robtarget pTarget_70:=[[1425.665446607,687.506980484,1450.952738403],[0.192522203,-0.943964264,-0.024409906,0.266965963],[-1,-1,-1,0],[9E+09,9E+09,9E+09,9E+09,9E+09,9E+09]];
    CONST robtarget pTarget_71:=[[1384.935237655,681.546156959,1451.40550961],[0.209990953,-0.937692069,-0.057329224,0.270833424],[-1,-1,-1,0],[9E+09,9E+09,9E+09,9E+09,9E+09,9E+09]];
    CONST robtarget pTarget_72:=[[1344.642694212,688.901204364,1445.68219623],[0.226216688,-0.931277455,-0.084280013,0.272846462],[-1,-1,-1,0],[9E+09,9E+09,9E+09,9E+09,9E+09,9E+09]];
    CONST robtarget pTarget_73:=[[1330.088366483,701.998985612,1439.718273795],[0.232359958,-0.929154019,-0.091650825,0.272546849],[-1,-1,-1,0],[9E+09,9E+09,9E+09,9E+09,9E+09,9E+09]];
    VAR syncident Ident_2;
    CONST robtarget pChange:=[[5143.454300106,0,1627.492950444],[0,0.923879533,0,0.382683432],[0,0,0,7],[9E+09,9E+09,9E+09,9E+09,9E+09,9E+09]];
!***********************************************************
    !
    ! Module:  Module1
    !
    ! Description:
    !   <Insert description here>
    !
    ! Author: ahmadk
    !
    ! Version: 1.0
    !
    !***********************************************************


    !***********************************************************
    !
    ! Procedure main
    !
    !   This is the entry point of your program
    !
    !***********************************************************
    PROC main()
        !Add your code here
    ENDPROC
    PROC mmPath_1()
        MoveJ p6700_Home,v1000,z100,tool0\WObj:=wobj0;
        SyncMoveOn Ident_1,Task_1;
        MoveJ pTarget_1\ID:=10,v1000,z100,tool0\WObj:=wobj0;
        MoveL pTarget_2\ID:=20,v1000,z100,tool0\WObj:=wobj0;
        MoveL pTarget_3\ID:=30,v1000,z100,tool0\WObj:=wobj0;
        MoveL pTarget_4\ID:=40,v1000,z100,tool0\WObj:=wobj0;
        MoveL pTarget_5\ID:=50,v1000,z100,tool0\WObj:=wobj0;
        MoveL pTarget_6\ID:=60,v1000,z100,tool0\WObj:=wobj0;
        MoveL pTarget_7\ID:=70,v1000,z100,tool0\WObj:=wobj0;
        MoveL pTarget_8\ID:=80,v1000,z100,tool0\WObj:=wobj0;
        MoveL pTarget_9\ID:=90,v1000,z100,tool0\WObj:=wobj0;
        MoveL pTarget_10\ID:=100,v1000,z100,tool0\WObj:=wobj0;
        MoveL pTarget_11\ID:=110,v1000,z100,tool0\WObj:=wobj0;
        MoveL pTarget_12\ID:=120,v1000,z100,tool0\WObj:=wobj0;
        MoveL pTarget_13\ID:=130,v1000,z100,tool0\WObj:=wobj0;
        MoveL pTarget_14\ID:=140,v1000,z100,tool0\WObj:=wobj0;
        MoveL pTarget_15\ID:=150,v1000,z100,tool0\WObj:=wobj0;
        MoveL pTarget_16\ID:=160,v1000,z100,tool0\WObj:=wobj0;
        MoveL pTarget_17\ID:=170,v1000,z100,tool0\WObj:=wobj0;
        MoveL pTarget_18\ID:=180,v1000,z100,tool0\WObj:=wobj0;
        MoveL pTarget_19\ID:=190,v1000,z100,tool0\WObj:=wobj0;
        MoveL pTarget_20\ID:=200,v1000,z100,tool0\WObj:=wobj0;
        MoveL pTarget_21\ID:=210,v1000,z100,tool0\WObj:=wobj0;
        MoveL pTarget_22\ID:=220,v1000,z100,tool0\WObj:=wobj0;
        MoveL pTarget_23\ID:=230,v1000,z100,tool0\WObj:=wobj0;
        MoveL pTarget_24\ID:=240,v1000,z100,tool0\WObj:=wobj0;
        MoveL pTarget_25\ID:=250,v1000,z100,tool0\WObj:=wobj0;
        MoveL pTarget_26\ID:=260,v1000,z100,tool0\WObj:=wobj0;
        MoveL pTarget_27\ID:=270,v1000,z100,tool0\WObj:=wobj0;
        MoveL pTarget_28\ID:=280,v1000,z100,tool0\WObj:=wobj0;
        MoveL pTarget_29\ID:=290,v1000,z100,tool0\WObj:=wobj0;
        MoveL pTarget_30\ID:=300,v1000,z100,tool0\WObj:=wobj0;
        MoveL pTarget_31\ID:=310,v1000,z100,tool0\WObj:=wobj0;
        MoveL pTarget_32\ID:=320,v1000,z100,tool0\WObj:=wobj0;
        MoveL pTarget_33\ID:=330,v1000,z100,tool0\WObj:=wobj0;
        MoveL pTarget_34\ID:=340,v1000,z100,tool0\WObj:=wobj0;
        MoveL pTarget_35\ID:=350,v1000,z100,tool0\WObj:=wobj0;
        MoveL pTarget_36\ID:=360,v1000,z100,tool0\WObj:=wobj0;
        MoveL pTarget_37\ID:=370,v1000,z100,tool0\WObj:=wobj0;
        MoveL pTarget_38\ID:=380,v1000,z100,tool0\WObj:=wobj0;
        MoveL pTarget_39\ID:=390,v1000,z100,tool0\WObj:=wobj0;
        MoveL pTarget_40\ID:=400,v1000,z100,tool0\WObj:=wobj0;
        MoveL pTarget_41\ID:=410,v1000,z100,tool0\WObj:=wobj0;
        MoveL pTarget_42\ID:=420,v1000,z100,tool0\WObj:=wobj0;
        MoveL pTarget_43\ID:=430,v1000,z100,tool0\WObj:=wobj0;
        MoveL pTarget_44\ID:=440,v1000,z100,tool0\WObj:=wobj0;
        MoveL pTarget_45\ID:=450,v1000,z100,tool0\WObj:=wobj0;
        MoveL pTarget_46\ID:=460,v1000,z100,tool0\WObj:=wobj0;
        MoveL pTarget_47\ID:=470,v1000,z100,tool0\WObj:=wobj0;
        MoveL pTarget_48\ID:=480,v1000,z100,tool0\WObj:=wobj0;
        MoveL pTarget_49\ID:=490,v1000,z100,tool0\WObj:=wobj0;
        MoveL pTarget_50\ID:=500,v1000,z100,tool0\WObj:=wobj0;
        MoveL pTarget_51\ID:=510,v1000,z100,tool0\WObj:=wobj0;
        MoveL pTarget_52\ID:=520,v1000,z100,tool0\WObj:=wobj0;
        MoveL pTarget_53\ID:=530,v1000,z100,tool0\WObj:=wobj0;
        MoveL pTarget_54\ID:=540,v1000,z100,tool0\WObj:=wobj0;
        MoveL pTarget_55\ID:=550,v1000,z100,tool0\WObj:=wobj0;
        MoveL pTarget_56\ID:=560,v1000,z100,tool0\WObj:=wobj0;
        MoveL pTarget_57\ID:=570,v1000,z100,tool0\WObj:=wobj0;
        MoveL pTarget_58\ID:=580,v1000,z100,tool0\WObj:=wobj0;
        MoveL pTarget_59\ID:=590,v1000,z100,tool0\WObj:=wobj0;
        MoveL pTarget_60\ID:=600,v1000,z100,tool0\WObj:=wobj0;
        MoveL pTarget_61\ID:=610,v1000,z100,tool0\WObj:=wobj0;
        MoveL pTarget_62\ID:=620,v1000,z100,tool0\WObj:=wobj0;
        MoveL pTarget_63\ID:=630,v1000,z100,tool0\WObj:=wobj0;
        MoveL pTarget_64\ID:=640,v1000,z100,tool0\WObj:=wobj0;
        MoveL pTarget_65\ID:=650,v1000,z100,tool0\WObj:=wobj0;
        MoveL pTarget_66\ID:=660,v1000,z100,tool0\WObj:=wobj0;
        MoveL pTarget_67\ID:=670,v1000,z100,tool0\WObj:=wobj0;
        MoveL pTarget_68\ID:=680,v1000,z100,tool0\WObj:=wobj0;
        MoveL pTarget_69\ID:=690,v1000,z100,tool0\WObj:=wobj0;
        MoveL pTarget_70\ID:=700,v1000,z100,tool0\WObj:=wobj0;
        MoveL pTarget_71\ID:=710,v1000,z100,tool0\WObj:=wobj0;
        MoveL pTarget_72\ID:=720,v1000,z100,tool0\WObj:=wobj0;
        MoveL pTarget_73\ID:=730,v1000,fine,tool0\WObj:=wobj0;
        SyncMoveOff Ident_2;
        MoveJ p6700_Home,v1000,z100,tool0\WObj:=wobj0;
        MoveJ pChange,v1000,z100,tool0\WObj:=wobj0;
    ENDPROC
    PROC myMain()
        mmPath_1;
    ENDPROC
ENDMODULE

--- Backups/Controller5/RAPID/TASK2/PROGMOD/CalibData.mod ---
MODULE CalibData
    PERS tooldata tSpintec:=[TRUE,[[31.792631019,0,229.638935148],[0.945518576,0,0.325568154,0]],[3,[-51.132047978,0,99.657990242],[1,0,0,0],0,0,0]];
    TASK PERS wobjdata obWorkpiece:=[FALSE,FALSE,"ROB_1",[[965.75691978,1010,1860.622138946],[0.000000116,-0.25881769,-0.000000433,0.965926189]],[[-70.000166728,-1010,719.999567419],[0.707105789,-0.000000116,-0.707107773,-0.000000433]]];
ENDMODULE

--- Backups/Controller5/RAPID/TASK2/PROGMOD/Module1.mod ---
MODULE Module1
        CONST robtarget p1600_Home:=[[560.152901107,0,1233.935371403],[0,0.477158761,0,0.878817112],[0,0,2,0],[9E+09,9E+09,9E+09,9E+09,9E+09,9E+09]];
    VAR syncident Ident_1;
    PERS tasks Task_1{2}:=[["T_ROB1"],["T_ROB2"]];
    CONST robtarget pTarget_1:=[[-249.999367219,-2.759503933,70.911791319],[0.082627052,-0.189001665,0.896559115,0.391960322],[-1,0,2,0],[9E+09,9E+09,9E+09,9E+09,9E+09,9E+09]];
    CONST robtarget pTarget_2:=[[-272.860994804,33.003713337,109.273686321],[0.078888886,-0.183345526,0.900091869,0.387292639],[-1,0,2,0],[9E+09,9E+09,9E+09,9E+09,9E+09,9E+09]];
    CONST robtarget pTarget_3:=[[-293.909747151,69.703915361,146.790608764],[0.066447689,-0.162722707,0.911372094,0.372165194],[-1,0,2,0],[9E+09,9E+09,9E+09,9E+09,9E+09,9E+09]];
    CONST robtarget pTarget_4:=[[-309.049057288,104.287364252,178.817535141],[0.044488261,-0.119397612,0.929423604,0.346318884],[0,0,2,0],[9E+09,9E+09,9E+09,9E+09,9E+09,9E+09]];
    CONST robtarget pTarget_5:=[[-315.82436696,131.079185384,200.514549492],[0.018847209,-0.056496391,0.946916759,0.315913899],[0,0,2,0],[9E+09,9E+09,9E+09,9E+09,9E+09,9E+09]];
    CONST robtarget pTarget_6:=[[-316.949093873,142.442010103,208.738875508],[0.005635439,-0.017961808,0.953951582,0.299369328],[0,0,2,0],[9E+09,9E+09,9E+09,9E+09,9E+09,9E+09]];
    CONST robtarget pTarget_7:=[[-316.981336532,150.771457316,214.363656376],[0.00472652,-0.015856219,-0.958220782,-0.285550649],[0,0,2,0],[9E+09,9E+09,9E+09,9E+09,9E+09,9E+09]];
    CONST robtarget pTarget_8:=[[-316.204048535,159.553535577,219.906336386],[0.015917508,-0.05682374,-0.961261763,-0.269246205],[0,0,2,0],[9E+09,9E+09,9E+09,9E+09,9E+09,9E+09]];
    CONST robtarget pTarget_9:=[[-312.751266422,174.803616127,228.540118146],[0.032209123,-0.130949879,-0.962189752,-0.236654987],[0,0,2,0],[9E+09,9E+09,9E+09,9E+09,9E+09,9E+09]];
    CONST robtarget pTarget_10:=[[-304.928487553,193.590972725,237.35167523],[0.043068547,-0.216929266,-0.956567695,-0.189907974],[0,0,2,0],[9E+09,9E+09,9E+09,9E+09,9E+09,9E+09]];
    CONST robtarget pTarget_11:=[[-295.35254505,209.582414865,243.17789314],[0.042988124,-0.279779228,-0.947977395,-0.145651859],[0,0,2,0],[9E+09,9E+09,9E+09,9E+09,9E+09,9E+09]];
    CONST robtarget pTarget_12:=[[-283.89767317,224.89172178,247.2508217],[0.035173025,-0.328290116,-0.938550871,-0.100552084],[0,0,2,0],[9E+09,9E+09,9E+09,9E+09,9E+09,9E+09]];
    CONST robtarget pTarget_13:=[[-263.239275575,247.748070357,250.552666299],[0.014250971,-0.37796017,-0.925055022,-0.034874436],[0,0,2,0],[9E+09,9E+09,9E+09,9E+09,9E+09,9E+09]];
    CONST robtarget pTarget_14:=[[-240.980203403,269.118585414,250.90982541],[0.007976683,0.402341156,0.915275131,-0.018149404],[0,0,2,0],[9E+09,9E+09,9E+09,9E+09,9E+09,9E+09]];
    CONST robtarget pTarget_15:=[[-208.411538431,298.031041245,247.790506063],[0.034910793,0.408676536,0.908701592,-0.077628235],[0,0,2,0],[9E+09,9E+09,9E+09,9E+09,9E+09,9E+09]];
    CONST robtarget pTarget_16:=[[-176.050652943,326.808930331,241.226021251],[0.053503703,0.389404955,0.910952456,-0.125166922],[0,0,2,0],[9E+09,9E+09,9E+09,9E+09,9E+09,9E+09]];
    CONST robtarget pTarget_17:=[[-156.251547721,345.811133404,235.321691527],[0.059919365,0.36278175,0.917514208,-0.151547844],[0,0,2,0],[9E+09,9E+09,9E+09,9E+09,9E+09,9E+09]];
    CONST robtarget pTarget_18:=[[-137.911367006,365.728959049,228.015632898],[0.060848306,0.321409713,0.928490022,-0.175782705],[0,0,2,0],[9E+09,9E+09,9E+09,9E+09,9E+09,9E+09]];
    CONST robtarget pTarget_19:=[[-123.074825841,385.296017373,219.901370788],[0.055303407,0.265093219,0.942346678,-0.196595667],[0,0,2,0],[9E+09,9E+09,9E+09,9E+09,9E+09,9E+09]];
    CONST robtarget pTarget_20:=[[-112.483952008,403.752551203,211.51909834],[0.044543145,0.199537763,0.95536135,-0.213272783],[0,0,2,0],[9E+09,9E+09,9E+09,9E+09,9E+09,9E+09]];
    CONST robtarget pTarget_21:=[[-105.66911776,420.539983076,203.415477486],[0.032817077,0.140384123,0.963573356,-0.225259238],[0,0,2,0],[9E+09,9E+09,9E+09,9E+09,9E+09,9E+09]];
    CONST robtarget pTarget_22:=[[-101.152730173,437.795026941,194.70341226],[0.02007137,0.08291124,0.968380047,-0.234441785],[0,0,2,0],[9E+09,9E+09,9E+09,9E+09,9E+09,9E+09]];
    CONST robtarget pTarget_23:=[[-99.0040493,453.549567144,186.489814416],[0.008561695,0.034579383,0.970065446,-0.240216557],[0,0,1,0],[9E+09,9E+09,9E+09,9E+09,9E+09,9E+09]];
    CONST robtarget pTarget_24:=[[-98.516394989,465.109909633,180.348088014],[0.000491395,0.001966291,0.970025575,-0.242994396],[0,0,1,0],[9E+09,9E+09,9E+09,9E+09,9E+09,9E+09]];
    CONST robtarget pTarget_25:=[[-98.913820285,477.215623072,173.84543664],[0.007456826,0.029529533,-0.969123936,0.244685919],[0,0,1,0],[9E+09,9E+09,9E+09,9E+09,9E+09,9E+09]];
    CONST robtarget pTarget_26:=[[-101.158760793,495.694459859,163.84647429],[0.018390599,0.072530228,-0.966611976,0.245076395],[0,0,1,0],[9E+09,9E+09,9E+09,9E+09,9E+09,9E+09]];
    CONST robtarget pTarget_27:=[[-106.104979829,517.566463562,152.024862353],[0.029263347,0.116194115,-0.962734999,0.242453924],[0,0,1,0],[9E+09,9E+09,9E+09,9E+09,9E+09,9E+09]];
    CONST robtarget pTarget_28:=[[-113.660346961,540.614341097,139.758405519],[0.038221783,0.154953239,-0.958456095,0.236411725],[0,-1,1,0],[9E+09,9E+09,9E+09,9E+09,9E+09,9E+09]];
    CONST robtarget pTarget_29:=[[-130.507549693,578.661351825,120.440667817],[0.047524101,0.206136989,-0.952386495,0.2195654],[0,-1,1,0],[9E+09,9E+09,9E+09,9E+09,9E+09,9E+09]];
    CONST robtarget pTarget_30:=[[-151.266393323,615.999238015,103.277260281],[0.050249688,0.24477104,-0.948497911,0.194714713],[0,-1,1,0],[9E+09,9E+09,9E+09,9E+09,9E+09,9E+09]];
    CONST robtarget pTarget_31:=[[-176.02610459,654.710741932,88.198539481],[0.046456986,0.275583142,-0.946795556,0.159605309],[0,-1,1,0],[9E+09,9E+09,9E+09,9E+09,9E+09,9E+09]];
    CONST robtarget pTarget_32:=[[-202.970542535,693.300547015,76.716257128],[0.035884116,0.297986116,-0.947053887,0.114041831],[0,-1,1,0],[9E+09,9E+09,9E+09,9E+09,9E+09,9E+09]];
    CONST robtarget pTarget_33:=[[-231.602130589,732.417304287,69.542021834],[0.018589095,0.31143545,-0.948397291,0.056612584],[0,-1,1,0],[9E+09,9E+09,9E+09,9E+09,9E+09,9E+09]];
    CONST robtarget pTarget_34:=[[-260.470210824,771.255251336,67.256102726],[0.000027118,0.313521967,-0.949580944,0.000077659],[0,-1,1,0],[9E+09,9E+09,9E+09,9E+09,9E+09,9E+09]];
    CONST robtarget pTarget_35:=[[-291.671653455,813.968299538,69.78080258],[0.017514958,-0.303598774,0.9510575,0.054869325],[0,-1,1,0],[9E+09,9E+09,9E+09,9E+09,9E+09,9E+09]];
    CONST robtarget pTarget_36:=[[-321.100482584,856.495332628,76.875137674],[0.030055142,-0.282317538,0.953462043,0.101506791],[0,-1,1,0],[9E+09,9E+09,9E+09,9E+09,9E+09,9E+09]];
    CONST robtarget pTarget_37:=[[-347.608236851,898.755866406,87.798617829],[0.03661292,-0.250273308,0.957292518,0.140049279],[0,-1,1,0],[9E+09,9E+09,9E+09,9E+09,9E+09,9E+09]];
    CONST robtarget pTarget_38:=[[-370.0464549,940.669416672,101.810752862],[0.036758138,-0.206846372,0.962600213,0.171067961],[0,-1,1,0],[9E+09,9E+09,9E+09,9E+09,9E+09,9E+09]];
    CONST robtarget pTarget_39:=[[-386.422870207,979.737745125,117.176024402],[0.030820624,-0.15395644,0.968381142,0.193869719],[0,-1,1,0],[9E+09,9E+09,9E+09,9E+09,9E+09,9E+09]];
    CONST robtarget pTarget_40:=[[-397.441727713,1019.682361901,134.633461354],[0.01837918,-0.084776151,0.973609592,0.211091382],[0,-1,2,0],[9E+09,9E+09,9E+09,9E+09,9E+09,9E+09]];
    CONST robtarget pTarget_41:=[[-400.68526788,1043.112626972,145.490242444],[0.008067365,-0.036072035,0.975216982,0.218141154],[0,0,2,0],[9E+09,9E+09,9E+09,9E+09,9E+09,9E+09]];
    CONST robtarget pTarget_42:=[[-401.329476368,1057.285914809,152.218968855],[0.000811987,-0.00358584,0.975219049,0.221210962],[-1,0,2,0],[9E+09,9E+09,9E+09,9E+09,9E+09,9E+09]];
    CONST robtarget pTarget_43:=[[-400.962720054,1070.625724022,158.636236091],[0.006312666,-0.02754754,-0.974356125,-0.223229532],[-1,0,2,0],[9E+09,9E+09,9E+09,9E+09,9E+09,9E+09]];
    CONST robtarget pTarget_44:=[[-398.849530954,1089.506582954,167.817808857],[0.016104926,-0.069657841,-0.97181004,-0.224663442],[-1,0,2,0],[9E+09,9E+09,9E+09,9E+09,9E+09,9E+09]];
    CONST robtarget pTarget_45:=[[-394.29581823,1110.83283784,178.260483341],[0.026405516,-0.113854454,-0.967470561,-0.224367166],[-1,0,2,0],[9E+09,9E+09,9E+09,9E+09,9E+09,9E+09]];
    CONST robtarget pTarget_46:=[[-380.757667282,1149.008190868,196.879200033],[0.041846543,-0.182836175,-0.957495657,-0.219138923],[-1,0,2,0],[9E+09,9E+09,9E+09,9E+09,9E+09,9E+09]];
    CONST robtarget pTarget_47:=[[-357.502548238,1192.923255868,217.60212677],[0.053666998,-0.246019085,-0.94554354,-0.206256825],[-1,0,2,0],[9E+09,9E+09,9E+09,9E+09,9E+09,9E+09]];
    CONST robtarget pTarget_48:=[[-328.871131584,1234.786110626,235.983778233],[0.058387182,-0.291828294,-0.936135211,-0.187291352],[-1,0,2,0],[9E+09,9E+09,9E+09,9E+09,9E+09,9E+09]];
    CONST robtarget pTarget_49:=[[-297.082202513,1274.587810161,251.518415059],[0.056709338,-0.324130465,-0.930183001,-0.162736218],[-1,0,2,0],[9E+09,9E+09,9E+09,9E+09,9E+09,9E+09]];
    CONST robtarget pTarget_50:=[[-262.487169544,1314.071354306,264.397885002],[0.048966326,-0.346373772,-0.92759546,-0.131126548],[-1,0,2,0],[9E+09,9E+09,9E+09,9E+09,9E+09,9E+09]];
    CONST robtarget pTarget_51:=[[-226.575198444,1353.203760165,273.991191603],[0.03530716,-0.35871904,-0.92829236,-0.091363833],[-1,0,2,0],[9E+09,9E+09,9E+09,9E+09,9E+09,9E+09]];
    CONST robtarget pTarget_52:=[[-190.835454984,1391.952044842,279.667338403],[0.016347916,-0.360036739,-0.931834961,-0.042307189],[-1,0,2,0],[9E+09,9E+09,9E+09,9E+09,9E+09,9E+09]];
    CONST robtarget pTarget_53:=[[-154.17832425,1433.250752389,280.669165784],[0.008033429,0.346250872,0.937854953,-0.021768907],[-1,0,2,0],[9E+09,9E+09,9E+09,9E+09,9E+09,9E+09]];
    CONST robtarget pTarget_54:=[[-136.486757318,1454.463382029,278.844216812],[0.02093735,0.331543339,0.941332059,-0.059452467],[0,0,2,0],[9E+09,9E+09,9E+09,9E+09,9E+09,9E+09]];
    CONST robtarget pTarget_55:=[[-119.667994947,1475.942313909,275.183061704],[0.033064953,0.31046011,0.944668189,-0.100614324],[0,0,2,0],[9E+09,9E+09,9E+09,9E+09,9E+09,9E+09]];
    CONST robtarget pTarget_56:=[[-95.23421766,1510.929497189,264.90036064],[0.047328965,0.26196812,0.948558033,-0.171377746],[0,0,2,0],[9E+09,9E+09,9E+09,9E+09,9E+09,9E+09]];
    CONST robtarget pTarget_57:=[[-75.879163631,1544.775316833,249.92732557],[0.048387235,0.203046981,0.951330794,-0.226716385],[0,0,2,0],[9E+09,9E+09,9E+09,9E+09,9E+09,9E+09]];
    CONST robtarget pTarget_58:=[[-61.453751357,1578.969573233,230.891791828],[0.037712511,0.135799258,0.953915563,-0.264917773],[0,0,2,0],[9E+09,9E+09,9E+09,9E+09,9E+09,9E+09]];
    CONST robtarget pTarget_59:=[[-52.709355316,1614.593121608,208.283153837],[0.017684195,0.058897435,0.955941718,-0.287043189],[0,0,2,0],[9E+09,9E+09,9E+09,9E+09,9E+09,9E+09]];
    CONST robtarget pTarget_60:=[[-50.934699689,1632.587258186,196.277463107],[0.006063338,0.019886972,0.956307978,-0.291620979],[0,0,2,0],[9E+09,9E+09,9E+09,9E+09,9E+09,9E+09]];
    CONST robtarget pTarget_61:=[[-50.774421373,1647.958649082,185.919783485],[0.003455043,0.011306726,-0.956305426,0.292130371],[0,0,2,0],[9E+09,9E+09,9E+09,9E+09,9E+09,9E+09]];
    CONST robtarget pTarget_62:=[[-52.135096903,1666.482081789,173.506543624],[0.014073891,0.04660989,-0.956181617,0.28869735],[0,0,2,0],[9E+09,9E+09,9E+09,9E+09,9E+09,9E+09]];
    CONST robtarget pTarget_63:=[[-58.784165359,1700.876830889,151.380550889],[0.030261256,0.106897681,-0.956235196,0.270686891],[0,0,1,0],[9E+09,9E+09,9E+09,9E+09,9E+09,9E+09]];
    CONST robtarget pTarget_64:=[[-65.575026565,1722.872557128,138.384921656],[0.037454996,0.142723783,-0.956661627,0.251048954],[0,0,1,0],[9E+09,9E+09,9E+09,9E+09,9E+09,9E+09]];
    CONST robtarget pTarget_65:=[[-74.174240255,1744.953068342,126.651812084],[0.041515823,0.176927532,-0.957346748,0.224633675],[0,0,1,0],[9E+09,9E+09,9E+09,9E+09,9E+09,9E+09]];
    CONST robtarget pTarget_66:=[[-84.218309667,1766.689454041,116.699308849],[0.041788008,0.208774714,-0.958068354,0.191760032],[0,0,1,0],[9E+09,9E+09,9E+09,9E+09,9E+09,9E+09]];
    CONST robtarget pTarget_67:=[[-95.705744302,1788.48102753,108.594683736],[0.037739774,0.238344582,-0.958506502,0.151765791],[0,-1,1,0],[9E+09,9E+09,9E+09,9E+09,9E+09,9E+09]];
    CONST robtarget pTarget_68:=[[-107.613651561,1808.886394545,102.938341083],[0.029652784,0.263007018,-0.958267247,0.108036583],[0,-1,1,0],[9E+09,9E+09,9E+09,9E+09,9E+09,9E+09]];
    CONST robtarget pTarget_69:=[[-120.621960396,1829.451402306,99.309687547],[0.017514553,0.28370735,-0.956929474,0.059070827],[0,-1,1,0],[9E+09,9E+09,9E+09,9E+09,9E+09,9E+09]];
    CONST robtarget pTarget_70:=[[-148.700181706,1869.906708876,98.057386407],[0.008453075,-0.309439943,0.950526698,0.025970423],[0,-1,1,0],[9E+09,9E+09,9E+09,9E+09,9E+09,9E+09]];
    CONST robtarget pTarget_71:=[[-178.288124099,1909.002656836,102.934665136],[0.030003932,-0.320093123,0.942777752,0.088375719],[0,-1,1,0],[9E+09,9E+09,9E+09,9E+09,9E+09,9E+09]];
    CONST robtarget pTarget_72:=[[-222.707062289,1964.208367066,117.387196058],[0.050888963,-0.321696598,0.933861387,0.147731248],[0,-1,1,0],[9E+09,9E+09,9E+09,9E+09,9E+09,9E+09]];
    CONST robtarget pTarget_73:=[[-250.000100712,1997.24045093,129.048804233],[0.058217616,-0.318394383,0.930737336,0.17018736],[0,-1,1,0],[9E+09,9E+09,9E+09,9E+09,9E+09,9E+09]];
    VAR syncident Ident_2;
!***********************************************************
    !
    ! Module:  Module1
    !
    ! Description:
    !   <Insert description here>
    !
    ! Author: ahmadk
    !
    ! Version: 1.0
    !
    !***********************************************************


    !***********************************************************
    !
    ! Procedure main
    !
    !   This is the entry point of your program
    !
    !***********************************************************
    PROC main()
        !Add your code here
    ENDPROC
    PROC mmPath_1()
        MoveJ p1600_Home,v1000,z100,tSpintec\WObj:=wobj0;
        SyncMoveOn Ident_1,Task_1;
        MoveJ pTarget_1\ID:=10,v200,z1,tSpintec\WObj:=obWorkpiece;
        MoveL pTarget_2\ID:=20,v200,z1,tSpintec\WObj:=obWorkpiece;
        MoveL pTarget_3\ID:=30,v200,z1,tSpintec\WObj:=obWorkpiece;
        MoveL pTarget_4\ID:=40,v200,z1,tSpintec\WObj:=obWorkpiece;
        MoveL pTarget_5\ID:=50,v200,z1,tSpintec\WObj:=obWorkpiece;
        MoveL pTarget_6\ID:=60,v200,z1,tSpintec\WObj:=obWorkpiece;
        MoveL pTarget_7\ID:=70,v200,z1,tSpintec\WObj:=obWorkpiece;
        MoveL pTarget_8\ID:=80,v200,z1,tSpintec\WObj:=obWorkpiece;
        MoveL pTarget_9\ID:=90,v200,z1,tSpintec\WObj:=obWorkpiece;
        MoveL pTarget_10\ID:=100,v200,z1,tSpintec\WObj:=obWorkpiece;
        MoveL pTarget_11\ID:=110,v200,z1,tSpintec\WObj:=obWorkpiece;
        MoveL pTarget_12\ID:=120,v200,z1,tSpintec\WObj:=obWorkpiece;
        MoveL pTarget_13\ID:=130,v200,z1,tSpintec\WObj:=obWorkpiece;
        MoveL pTarget_14\ID:=140,v200,z1,tSpintec\WObj:=obWorkpiece;
        MoveL pTarget_15\ID:=150,v200,z1,tSpintec\WObj:=obWorkpiece;
        MoveL pTarget_16\ID:=160,v200,z1,tSpintec\WObj:=obWorkpiece;
        MoveL pTarget_17\ID:=170,v200,z1,tSpintec\WObj:=obWorkpiece;
        MoveL pTarget_18\ID:=180,v200,z1,tSpintec\WObj:=obWorkpiece;
        MoveL pTarget_19\ID:=190,v200,z1,tSpintec\WObj:=obWorkpiece;
        MoveL pTarget_20\ID:=200,v200,z1,tSpintec\WObj:=obWorkpiece;
        MoveL pTarget_21\ID:=210,v200,z1,tSpintec\WObj:=obWorkpiece;
        MoveL pTarget_22\ID:=220,v200,z1,tSpintec\WObj:=obWorkpiece;
        MoveL pTarget_23\ID:=230,v200,z1,tSpintec\WObj:=obWorkpiece;
        MoveL pTarget_24\ID:=240,v200,z1,tSpintec\WObj:=obWorkpiece;
        MoveL pTarget_25\ID:=250,v200,z1,tSpintec\WObj:=obWorkpiece;
        MoveL pTarget_26\ID:=260,v200,z1,tSpintec\WObj:=obWorkpiece;
        MoveL pTarget_27\ID:=270,v200,z1,tSpintec\WObj:=obWorkpiece;
        MoveL pTarget_28\ID:=280,v200,z1,tSpintec\WObj:=obWorkpiece;
        MoveL pTarget_29\ID:=290,v200,z1,tSpintec\WObj:=obWorkpiece;
        MoveL pTarget_30\ID:=300,v200,z1,tSpintec\WObj:=obWorkpiece;
        MoveL pTarget_31\ID:=310,v200,z1,tSpintec\WObj:=obWorkpiece;
        MoveL pTarget_32\ID:=320,v200,z1,tSpintec\WObj:=obWorkpiece;
        MoveL pTarget_33\ID:=330,v200,z1,tSpintec\WObj:=obWorkpiece;
        MoveL pTarget_34\ID:=340,v200,z1,tSpintec\WObj:=obWorkpiece;
        MoveL pTarget_35\ID:=350,v200,z1,tSpintec\WObj:=obWorkpiece;
        MoveL pTarget_36\ID:=360,v200,z1,tSpintec\WObj:=obWorkpiece;
        MoveL pTarget_37\ID:=370,v200,z1,tSpintec\WObj:=obWorkpiece;
        MoveL pTarget_38\ID:=380,v200,z1,tSpintec\WObj:=obWorkpiece;
        MoveL pTarget_39\ID:=390,v200,z1,tSpintec\WObj:=obWorkpiece;
        MoveL pTarget_40\ID:=400,v200,z1,tSpintec\WObj:=obWorkpiece;
        MoveL pTarget_41\ID:=410,v200,z1,tSpintec\WObj:=obWorkpiece;
        MoveL pTarget_42\ID:=420,v200,z1,tSpintec\WObj:=obWorkpiece;
        MoveL pTarget_43\ID:=430,v200,z1,tSpintec\WObj:=obWorkpiece;
        MoveL pTarget_44\ID:=440,v200,z1,tSpintec\WObj:=obWorkpiece;
        MoveL pTarget_45\ID:=450,v200,z1,tSpintec\WObj:=obWorkpiece;
        MoveL pTarget_46\ID:=460,v200,z1,tSpintec\WObj:=obWorkpiece;
        MoveL pTarget_47\ID:=470,v200,z1,tSpintec\WObj:=obWorkpiece;
        MoveL pTarget_48\ID:=480,v200,z1,tSpintec\WObj:=obWorkpiece;
        MoveL pTarget_49\ID:=490,v200,z1,tSpintec\WObj:=obWorkpiece;
        MoveL pTarget_50\ID:=500,v200,z1,tSpintec\WObj:=obWorkpiece;
        MoveL pTarget_51\ID:=510,v200,z1,tSpintec\WObj:=obWorkpiece;
        MoveL pTarget_52\ID:=520,v200,z1,tSpintec\WObj:=obWorkpiece;
        MoveL pTarget_53\ID:=530,v200,z1,tSpintec\WObj:=obWorkpiece;
        MoveL pTarget_54\ID:=540,v200,z1,tSpintec\WObj:=obWorkpiece;
        MoveL pTarget_55\ID:=550,v200,z1,tSpintec\WObj:=obWorkpiece;
        MoveL pTarget_56\ID:=560,v200,z1,tSpintec\WObj:=obWorkpiece;
        MoveL pTarget_57\ID:=570,v200,z1,tSpintec\WObj:=obWorkpiece;
        MoveL pTarget_58\ID:=580,v200,z1,tSpintec\WObj:=obWorkpiece;
        MoveL pTarget_59\ID:=590,v200,z1,tSpintec\WObj:=obWorkpiece;
        MoveL pTarget_60\ID:=600,v200,z1,tSpintec\WObj:=obWorkpiece;
        MoveL pTarget_61\ID:=610,v200,z1,tSpintec\WObj:=obWorkpiece;
        MoveL pTarget_62\ID:=620,v200,z1,tSpintec\WObj:=obWorkpiece;
        MoveL pTarget_63\ID:=630,v200,z1,tSpintec\WObj:=obWorkpiece;
        MoveL pTarget_64\ID:=640,v200,z1,tSpintec\WObj:=obWorkpiece;
        MoveL pTarget_65\ID:=650,v200,z1,tSpintec\WObj:=obWorkpiece;
        MoveL pTarget_66\ID:=660,v200,z1,tSpintec\WObj:=obWorkpiece;
        MoveL pTarget_67\ID:=670,v200,z1,tSpintec\WObj:=obWorkpiece;
        MoveL pTarget_68\ID:=680,v200,z1,tSpintec\WObj:=obWorkpiece;
        MoveL pTarget_69\ID:=690,v200,z1,tSpintec\WObj:=obWorkpiece;
        MoveL pTarget_70\ID:=700,v200,z1,tSpintec\WObj:=obWorkpiece;
        MoveL pTarget_71\ID:=710,v200,z1,tSpintec\WObj:=obWorkpiece;
        MoveL pTarget_72\ID:=720,v200,z1,tSpintec\WObj:=obWorkpiece;
        MoveL pTarget_73\ID:=730,v200,fine,tSpintec\WObj:=obWorkpiece;
        SyncMoveOff Ident_2;
        MoveJ p1600_Home,v1000,z100,tSpintec\WObj:=wobj0;
    ENDPROC
    PROC myMain()
        mmPath_1;
    ENDPROC
ENDMODULE
